{attribute 'linkalways'} 
{attribute 'no_explicit_call' := 'This FB is a CLASS and must be accessed using methods or properties'}
{attribute 'enable_dynamic_creation'}
FUNCTION_BLOCK MockAliasDatatype_HRESULT EXTENDS AliasDatatypeBase
VAR
	localData : HRESULT;
	activeData : REFERENCE TO HRESULT REF= localData;
	aliasBaseDatatype : _DINT(localData);
END_VAR

PROPERTY PUBLIC Address : PVOID
GET
Address := ADR(activeData);
END_GET
END_PROPERTY

METHOD PUBLIC ClearReference
VAR_INPUT
END_VAR
activeData REF= localData;
SetBaseDatatypeReference();
END_METHOD

METHOD PUBLIC Clone : I_Datatype
VAR
    pClone : POINTER TO MockAliasDatatype_HRESULT;
END_VAR
pClone := __NEW(MockAliasDatatype_HRESULT(InitialValue := Value));
Clone := pClone^;
END_METHOD

METHOD FB_init : BOOL
VAR_INPUT
	bInitRetains : BOOL; // if TRUE, the retain variables are initialized (warm start / cold start)
	bInCopyCode : BOOL;  // if TRUE, the instance afterwards gets moved into the copy code (online change)
	InitialValue : HRESULT;
END_VAR
localData := InitialValue;
SetBaseDatatypeReference();
AddBaseDatatype(aliasBaseDatatype);
END_METHOD

PROPERTY PUBLIC Identifier : T_MAXSTRING
GET
Identifier := 'HRESULT';
END_GET
END_PROPERTY

METHOD PUBLIC MakeReferenceTo
VAR_INPUT
	ReferenceTarget : REFERENCE TO HRESULT;
END_VAR
activeData REF= ReferenceTarget;
SetBaseDatatypeReference();
END_METHOD

METHOD PROTECTED SetBaseDatatypeReference
VAR_INPUT
END_VAR
aliasBaseDatatype.MakeReferenceTo(activeData);
END_METHOD

PROPERTY PUBLIC Size : UDINT
GET
Size := SIZEOF(activeData);
END_GET
END_PROPERTY

METHOD TryMakeReferenceTo : BOOL
VAR_INPUT
	Target : I_Datatype;
END_VAR
VAR
	targetAsAlias : I_AliasDatatype;
	pTargetData : POINTER TO HRESULT;
END_VAR
IF NOT Target.TryResolveAsAliasDatatype(targetAsAlias) THEN
	RETURN;
END_IF

IF targetAsAlias.Identifier <> Identifier THEN
	RETURN;
END_IF

pTargetData := Target.Address;
activeData REF= pTargetData^;
SetBaseDatatypeReference();
TryMakeReferenceTo := TRUE;
END_METHOD

PROPERTY PUBLIC Value : REFERENCE TO HRESULT
GET
Value REF= activeData;
END_GET
END_PROPERTY

END_FUNCTION_BLOCK

(* stored: Version 1.1.0.1, ProductVersion 3.1.4024.12
   POU MockAliasDatatype_HRESULT: Id {72a17a98-cc7f-49ef-9dd3-ffb7be4e211a}, SpecialFunc None
   Folder Constructor: Id {de40222d-6778-459a-bb19-4254012ad3da}
   Folder Protected: Id {207d39dd-beb6-487d-92f7-8fb014a1653d}
   Property Address: Id {dfb60c57-b0a6-4be3-8cfc-737df02bca39}
   Get Get: Id {83932da7-808b-4eae-bc5d-bcbb0d6f602c}
   Method ClearReference: Id {3f2d0897-1169-45d0-b5b7-ec342beb91b8}
   Method Clone: Id {8d3523ad-19f9-44d1-af8c-47f88cffa8fa}
   Method FB_init: Id {99f15046-4899-41b2-ac3d-1e85d75b1d35}
   Property Identifier: Id {c1ca2e72-5b34-48af-abab-a4da689999a0}
   Get Get: Id {11e0a0e1-6bf1-41c1-b186-96098d982a16}
   Method MakeReferenceTo: Id {897bf8fa-b6da-4451-bdac-0383e9264852}
   Method SetBaseDatatypeReference: Id {973aaacc-b431-45d7-bcda-e425ee4dd0ef}
   Property Size: Id {af7c3aa7-35af-4023-95b3-bb905e3e50b2}
   Get Get: Id {63e6a7d7-a4a1-41e2-ab35-f717c3866c4e}
   Method TryMakeReferenceTo: Id {4e30d1a9-a1d0-4537-ab05-3d5644f69d0e}
   Property Value: Id {66a95d13-bcd7-45da-8840-f91e6a4bd783}
   Get Get: Id {a32f3b0e-b8ff-4b54-8e11-c9c7a479cf0d} *)
